PROGRAM Signal1
VAR
	fbTimer1: TON;			//Timer1 Initialization
	fbTimer2: TON;			//Timer2 Initialization
	Blinker: FB_Blinker1;	//Function Block Blinker1 Initialization
END_VAR

//Timer1 Parameterization
fbTimer1(IN := GVL_Var.bCompressor,
		PT	:= GVL_Var.tlmAlaramThreshold,
		Q	=> GVL_Var.bSignal
		);
//Timer2 Parameterization
fbTimer2(IN := GVL_Var.bDoorOpen,
		PT	:= GVL_Var.tlmAlaramThreshold
		);
//Blinker Parameterization	
Blinker(bStart := fbTimer2.Q,
		tSignalTimeOff := T#1S, 
		tSignalTimeOn	:= T#1S,
		bOut => GVL_Var.bSignal );
//To switch ON the Lamp when Door is open		
IF GVL_Var.bDoorOpen THEN
	GVL_Var.bLamp := TRUE;
ELSIF NOT GVL_Var.bDoorOpen THEN
	GVL_Var.bLamp := FALSE;
END_IF

END_PROGRAM

(* stored: Version 1.1.0.1, ProductVersion 3.1.4024.4
   POU Signal1: Id {1523f310-75c7-4178-a880-46a717c37a5c}, SpecialFunc None *)
